TYPE TcaWorkpiecePlaceData : 
STRUCT
	Enabled : BOOL; // tot wird nicht mehr benötigt
	Id : INT;	// <> 0 Workpiece Present 
	Error : BOOL;
	SerialNumber : STRING;
	CurrentStatus : eTcaWorkpiecePlaceStatus;
	RequestStatus : eTcaWorkpiecePlaceStatus;
	Shape : eTcaWorkpiecePlaceShape;
	Volume : ST_Coordinate;
	Logging : WSTRING;	// Information in csv, xml or json Format
	
	
END_STRUCT
END_TYPE

(* stored: Version 1.1.0.1
   DUT TcaWorkpiecePlaceData: Id {7ca366c4-6112-4745-8034-11405d12e349} *)
